PROGRAM MAIN
VAR
	stRoomCheckDefaultParameters : ST_RangeCheckDefaultParameters := (tTaskCycleTime := GlobalVariables.tCtrlCycleTime_MAIN, tCtrlCycleTime := GlobalVariables.tCtrlCycleTime_MAIN, fRestoreDifference := 4);
	Room_Check : FB_RangeCheck := (ST_DefaultParameters := stRoomCheckDefaultParameters);
	
	Ambient : FB_Ambient;
	BufferStorage : FB_BufferStorage;
	ActiveWallModules : FB_ActiveWallModulesSystem;
	AirHandlingUnit : FB_AirHandlingUnitSystem;
	CN : FB_CNSystem;
	HNLT: FB_HNLTSystem;
	
	PCH : FB_PowerControlledHeaterSystem;
END_VAR

Ambient();
BufferStorage();

//set algorithm permission depending on production mode to control structs
Room_Check(fInput := Ambient.localState.fRoomTemperature,
	fLowerLimit := 5,
	fUpperLimit := 30);

ActiveWallModules(bSetStatusOnAutomatic := FALSE,
	fSetPointAutomatic := 0,
	bAlgorithmPermission := Room_Check.bPermission,
	bHeatingModeAutomatic := FALSE,
	fHysteresisRangeAutomatic := 3,
	stAmbientState := Ambient.localState);
	
AirHandlingUnit(bSetStatusOnAutomatic := FALSE,
	fSetPointAutomatic := 0,
	bAlgorithmPermission := Room_Check.bPermission,
	bHeatingModeAutomatic := FALSE,
	fHysteresisRangeAutomatic := 3,
	stAmbientState := Ambient.localState);
	
CN(bSetStatusOnAutomatic := FALSE,
	fSetPointAutomatic := 0,
	bAlgorithmPermission := Room_Check.bPermission);

HNLT();	
	
PCH(bSetStatusOnAutomatic := FALSE,
	bAlgorithmPermission := Room_Check.bPermission,
	fSetPointAutomatic := 0);

END_PROGRAM

(* stored: Version 1.1.0.1, ProductVersion 3.1.4024.6
   POU MAIN: Id {9962e183-3753-4780-b1ab-bc2415940cfb}, SpecialFunc None *)
